// TIA Portal V18 export
DATA_BLOCK "ServoV90_A2"   // DB2502
{ S7_Optimized_Access := 'FALSE' }
// stored: AutoNumber false
   VAR
      In : Struct
         iInterlock : Bool;   // interlock
         "iManJog+" : Bool;   // positive motion/action/...manually
         "iManJog-" : Bool;   // negtive motion/action/...manually
         iAutoStart : Bool;   // negtive motion/action/...automaticly
         iHome : Bool;   // Homing
         iCancelTask : Bool;   // Cancel task
         iPauseTask : Bool;   // Pause task
         iManStart : Bool;   // positive motion/action/...automaticly
         iManListStart : Bool;
         iLimitSwitchActive : Bool;
         iLimitSoftActive : Bool;
         iRunningTimeout : Time;
         iHomingTimeout : Time;
         iAutoPosition : DInt;
         iAutoVelocity : Int;
         iManListPosition : DInt;
         iManListVelocity : Int;
         iManListNumber : Int;   // position list number
         iManPosition : DInt;
         iManVelocity : Int;
         iMode : Int;   // 1-相对;2-绝对
      END_STRUCT;
      Out : Struct
         oReady : Bool;
         oWarning : Bool;   // warning
         oError : Bool;   // error
         oInterlock : Bool;
         oServoEnable : Bool;
         oRunning : Bool;
         oHoming : Bool;
         oHomeRef : Bool;
         oServoPosOK : Bool;
         oErrorCode : Int;
         oStatus : Int;
         oActPosition : DInt;
         oManualListPos : DInt;
      END_STRUCT;
      IO : Struct
         ioManEnale : Bool;
         ioAutoEnale : Bool;
      END_STRUCT;
      Spare : Struct
         S : Array[0..100] of Byte;
      END_STRUCT;
      Manual : Struct
         Index : Int := 1;
         Pos : Array[1..20] of Struct
            Pos : DInt;
            Vel : Int;
         END_STRUCT;
      END_STRUCT;
      Auto : Struct
         Index : Int := 1;
         Pos : Array[1..20] of Struct
            Pos : DInt;
            Vel : Int;
         END_STRUCT;
      END_STRUCT;
      Interlock : Struct
         Active : Bool := FALSE;
         Case1 : Bool := TRUE;
         Case2 : Bool := TRUE;
         Case3 : Bool := FALSE;
         Case4 : Bool := FALSE;
         Case5 : Bool := FALSE;
         Case6 : Bool := FALSE;
         Case7 : Bool := FALSE;
         Case8 : Bool := FALSE;
         Case9 : Bool := FALSE;
         Case10 : Bool := FALSE;
      END_STRUCT;
      PositionOk : Array[1..20] of Bool;
      Home_Pos : Struct
         "Home Pos Pls" : Bool := FALSE;
         "Arrow indication" : Int := 0;
         "Process prompt" : Int := 0;
         "Button prompt" : Int := 0;
      END_STRUCT;
   END_VAR
BEGIN
   Spare.S[0..100] := 16#00;
   Manual.Pos[1].Pos := 0;
   Manual.Pos[2].Pos := 450000;
   Manual.Pos[3].Pos := 900000;
   Manual.Pos[4].Pos := 135000;
   Manual.Pos[5].Pos := 180000;
   Manual.Pos[6].Pos := 225000;
   Manual.Pos[7].Pos := 270000;
   Manual.Pos[8].Pos := 315000;
   Manual.Pos[9..20].Pos := 0;
   Manual.Pos[1..8].Vel := 10000;
   Manual.Pos[9..20].Vel := 0;
   Auto.Pos[1].Pos := 0;
   Auto.Pos[2].Pos := 450000;
   Auto.Pos[3].Pos := 900000;
   Auto.Pos[4].Pos := 135000;
   Auto.Pos[5].Pos := 180000;
   Auto.Pos[6].Pos := 225000;
   Auto.Pos[7].Pos := 270000;
   Auto.Pos[8].Pos := 315000;
   Auto.Pos[9..20].Pos := 0;
   Auto.Pos[1..8].Vel := 10000;
   Auto.Pos[9..20].Vel := 0;
   // Auto.Pos[1] : 1.取料位置
   // Auto.Pos[2] : 2.放料位置
   // Auto.Pos[3] : 3.
   // Auto.Pos[4] : 4.
   // Auto.Pos[5] : 5.
   // Auto.Pos[6] : 6.
   // Auto.Pos[7] : 7.
   // Auto.Pos[8] : 8.
   // Auto.Pos[9] : 9.
   PositionOk[1] := FALSE;   // [1]
   PositionOk[2] := FALSE;   // [2]
   PositionOk[3] := FALSE;   // [3]
   PositionOk[4] := FALSE;   // [4]
   PositionOk[5] := FALSE;   // [5]
   PositionOk[6] := FALSE;   // [6]
   PositionOk[7] := FALSE;   // [7]
   PositionOk[8] := FALSE;   // [8]
   PositionOk[9] := FALSE;   // [9]
   PositionOk[10..20] := FALSE;
END_DATA_BLOCK
